Omron Sysmac Studio project Shifting (Sysmac Studio 1.65.0.64007, StandardProject)

# Controller new_Controller_0: NX1P2-1040DT1 version 1.69
Task PrimaryTask (priority 4, period or condition 2000): Program0

VAR_GLOBAL
    IN_Start_But : BOOL;
    IN_Stop_But : BOOL;
    IN_Small_Sens : BOOL;
    IN_Medium_Sens : BOOL;
    IN_High_Sens : BOOL;
    OUT_Konveyor_Start : BOOL;
    OUT_Vana1 : BOOL;
    OUT_Vana2 : BOOL;
    OUT_Vana3 : BOOL;
    OUT_Vana4 : BOOL;
    OUT_Vana5 : BOOL;
    OUT_Vana6 : BOOL;
    OUT_Vana7 : BOOL;
    OUT_Vana8 : BOOL;
    Ary_Bottle : ARRAY[0..8] OF INT;
END_VAR

PROGRAM Program0
VAR
    Start : BOOL;
    Kutu : BOOL;
    Ton_Small : TON;
    medi : BOOL;
    Small_Bottle : BOOL;
    High_Bottle : BOOL;
    Medium_Bottle : BOOL;
    Big_Bottle : BOOL;
    Sayac : INT;
    OUT_Konveyor_Calis : BOOL;
    Konveyor_Calis : BOOL;
    TON_Konv : TON;
    Shiftle : BOOL;
    Small_Bottlei : BOOL;
    TON_Small_Dly : TON;
    TON_Medium_Dly : TON;
    TON_Big_Dly : TON;
    TON_Vana : TON;
    OUT_Vana : BOOL;
    Set_Small : BOOL;
    Set_Medium : BOOL;
    Set_Big : BOOL;
END_VAR
VAR_EXTERNAL
    IN_Start_But : BOOL;
    IN_Stop_But : BOOL;
    IN_Small_Sens : BOOL;
    IN_Medium_Sens : BOOL;
    IN_High_Sens : BOOL;
    OUT_Konveyor_Start : BOOL;
    Ary_Bottle : ARRAY[0..8] OF INT;
    OUT_Vana1 : BOOL;
    OUT_Vana2 : BOOL;
    OUT_Vana3 : BOOL;
    OUT_Vana4 : BOOL;
    OUT_Vana5 : BOOL;
    OUT_Vana6 : BOOL;
    OUT_Vana7 : BOOL;
    OUT_Vana8 : BOOL;
END_VAR
VAR
    _e1 : R_TRIG;
    _e2 : R_TRIG;
    _e3 : R_TRIG;
    _e4 : R_TRIG;
    _e5 : R_TRIG;
    _e6 : R_TRIG;
    _e7 : F_TRIG;
    _e8 : F_TRIG;
    _e9 : F_TRIG;
    _e10 : R_TRIG;
    _e11 : R_TRIG;
    _e12 : R_TRIG;
    _e13 : R_TRIG;
    _e14 : R_TRIG;
    _e15 : R_TRIG;
    _e16 : R_TRIG;
END_VAR

(* Section Section0: ladder, written here as Structured Text *)

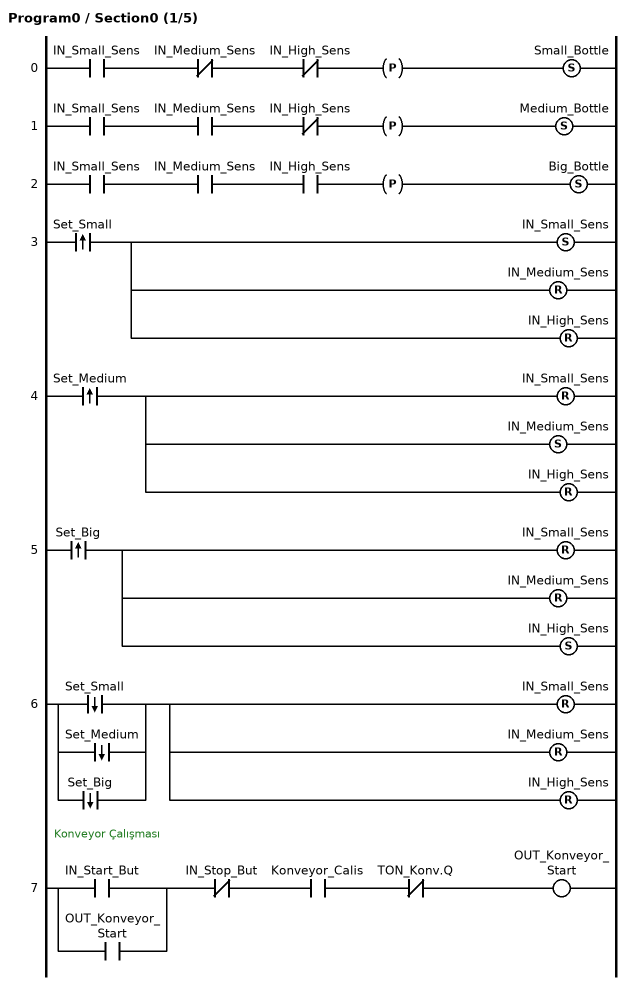
(* Rung 0 *)
_e1(CLK := IN_Small_Sens AND NOT IN_Medium_Sens AND NOT IN_High_Sens);
IF _e1.Q THEN Small_Bottle := TRUE; END_IF;
(* Rung 1 *)
_e2(CLK := IN_Small_Sens AND IN_Medium_Sens AND NOT IN_High_Sens);
IF _e2.Q THEN Medium_Bottle := TRUE; END_IF;
(* Rung 2 *)
_e3(CLK := IN_Small_Sens AND IN_Medium_Sens AND IN_High_Sens);
IF _e3.Q THEN Big_Bottle := TRUE; END_IF;
(* Rung 3 *)
_e4(CLK := Set_Small);
IF _e4.Q THEN
    IN_Small_Sens := TRUE;
    IN_Medium_Sens := FALSE;
    IN_High_Sens := FALSE;
END_IF;
(* Rung 4 *)
_e5(CLK := Set_Medium);
IF _e5.Q THEN
    IN_Small_Sens := FALSE;
    IN_Medium_Sens := TRUE;
    IN_High_Sens := FALSE;
END_IF;
(* Rung 5 *)
_e6(CLK := Set_Big);
IF _e6.Q THEN
    IN_Small_Sens := FALSE;
    IN_Medium_Sens := FALSE;
    IN_High_Sens := TRUE;
END_IF;
(* Rung 6 *)
_e7(CLK := Set_Small);
_e8(CLK := Set_Medium);
_e9(CLK := Set_Big);
IF _e7.Q OR _e8.Q OR _e9.Q THEN
    IN_Small_Sens := FALSE;
    IN_Medium_Sens := FALSE;
    IN_High_Sens := FALSE;
END_IF;
(* Rung 7: Konveyor Çalışması *)
OUT_Konveyor_Start := (IN_Start_But OR OUT_Konveyor_Start) AND NOT IN_Stop_But AND Konveyor_Calis AND NOT TON_Konv.Q;

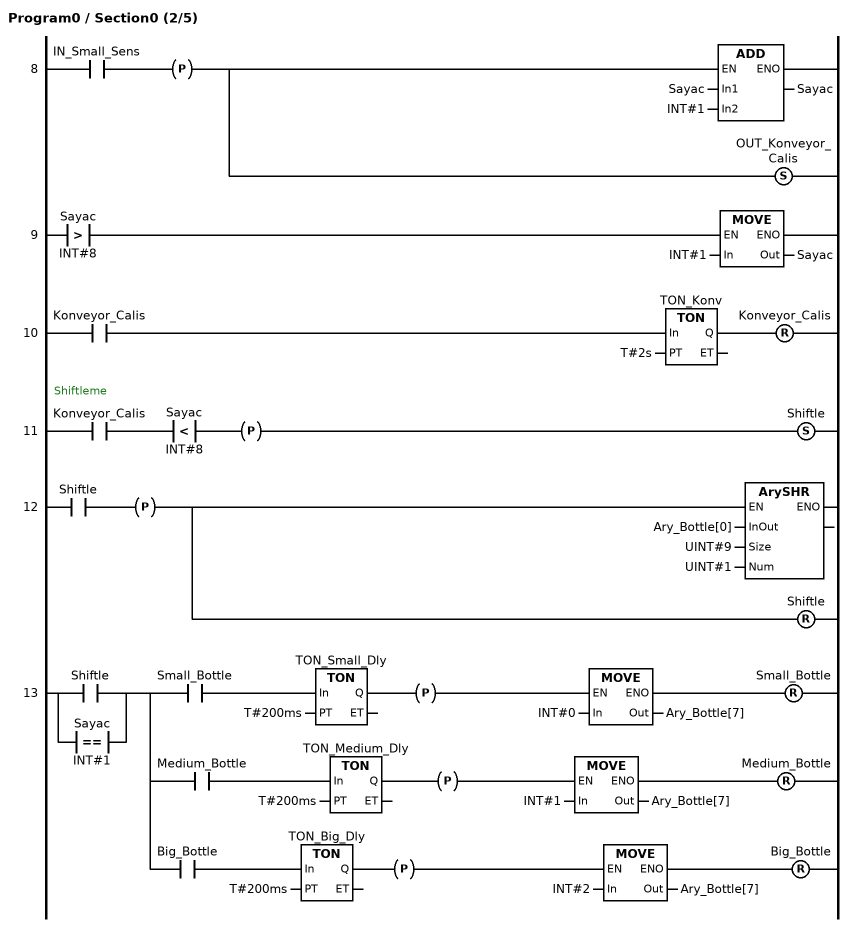
(* Rung 8 *)
_e10(CLK := IN_Small_Sens);
IF _e10.Q THEN
    Sayac := Sayac + INT#1;
    OUT_Konveyor_Calis := TRUE;
END_IF;
(* Rung 9 *)
IF Sayac > INT#8 THEN Sayac := INT#1; END_IF;
(* Rung 10 *)
TON_Konv(In := Konveyor_Calis, PT := T#2s);
IF TON_Konv.Q THEN Konveyor_Calis := FALSE; END_IF;
(* Rung 11: Shiftleme *)
_e11(CLK := Konveyor_Calis AND (Sayac < INT#8));
IF _e11.Q THEN Shiftle := TRUE; END_IF;
(* Rung 12 *)
_e12(CLK := Shiftle);
IF _e12.Q THEN
    ArySHR(InOut := Ary_Bottle[0], Size := UINT#9, Num := UINT#1);
    Shiftle := FALSE;
END_IF;
(* Rung 13 *)
TON_Small_Dly(In := (Shiftle OR (Sayac = INT#1)) AND Small_Bottle, PT := T#200ms);
_e13(CLK := TON_Small_Dly.Q);
IF _e13.Q THEN
    Ary_Bottle[7] := INT#0;
    Small_Bottle := FALSE;
END_IF;
TON_Medium_Dly(In := (Shiftle OR (Sayac = INT#1)) AND Medium_Bottle, PT := T#200ms);
_e14(CLK := TON_Medium_Dly.Q);
IF _e14.Q THEN
    Ary_Bottle[7] := INT#1;
    Medium_Bottle := FALSE;
END_IF;
TON_Big_Dly(In := (Shiftle OR (Sayac = INT#1)) AND Big_Bottle, PT := T#200ms);
_e15(CLK := TON_Big_Dly.Q);
IF _e15.Q THEN
    Ary_Bottle[7] := INT#2;
    Big_Bottle := FALSE;
END_IF;

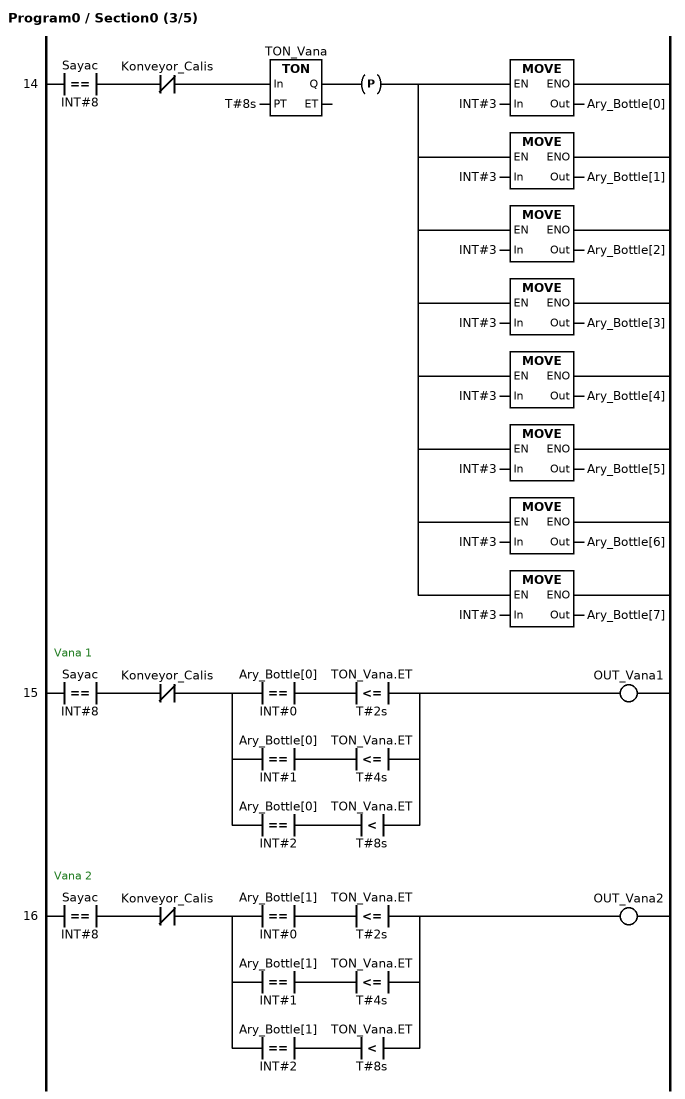
(* Rung 14 *)
TON_Vana(In := (Sayac = INT#8) AND NOT Konveyor_Calis, PT := T#8s);
_e16(CLK := TON_Vana.Q);
IF _e16.Q THEN
    Ary_Bottle[0] := INT#3;
    Ary_Bottle[1] := INT#3;
    Ary_Bottle[2] := INT#3;
    Ary_Bottle[3] := INT#3;
    Ary_Bottle[4] := INT#3;
    Ary_Bottle[5] := INT#3;
    Ary_Bottle[6] := INT#3;
    Ary_Bottle[7] := INT#3;
END_IF;
(* Rung 15: Vana 1 *)
OUT_Vana1 := (Sayac = INT#8) AND NOT Konveyor_Calis AND (((Ary_Bottle[0] = INT#0) AND (TON_Vana.ET <= T#2s)) OR ((Ary_Bottle[0] = INT#1) AND (TON_Vana.ET <= T#4s)) OR ((Ary_Bottle[0] = INT#2) AND (TON_Vana.ET < T#8s)));
(* Rung 16: Vana 2 *)
OUT_Vana2 := (Sayac = INT#8) AND NOT Konveyor_Calis AND (((Ary_Bottle[1] = INT#0) AND (TON_Vana.ET <= T#2s)) OR ((Ary_Bottle[1] = INT#1) AND (TON_Vana.ET <= T#4s)) OR ((Ary_Bottle[1] = INT#2) AND (TON_Vana.ET < T#8s)));

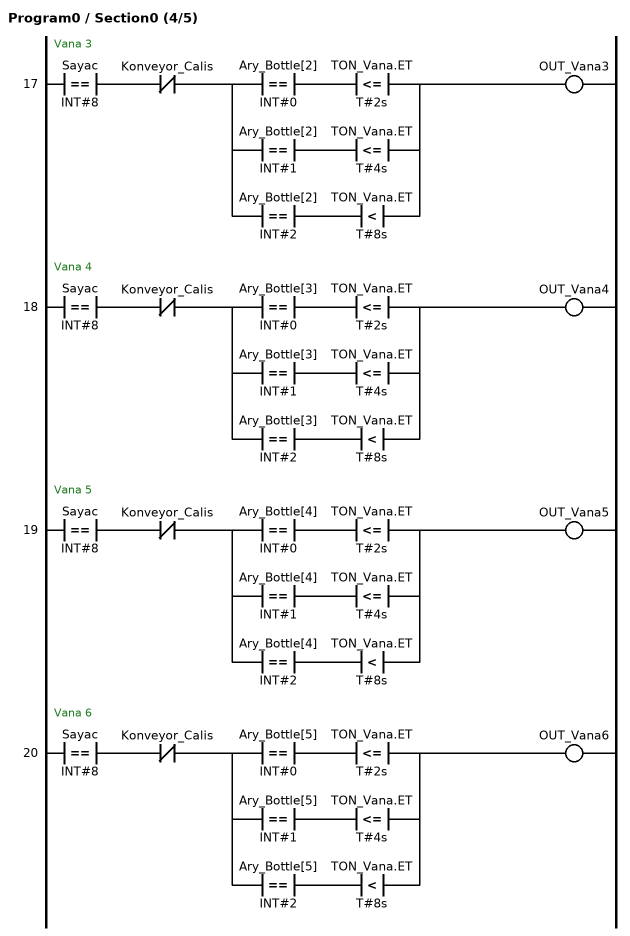
(* Rung 17: Vana 3 *)
OUT_Vana3 := (Sayac = INT#8) AND NOT Konveyor_Calis AND (((Ary_Bottle[2] = INT#0) AND (TON_Vana.ET <= T#2s)) OR ((Ary_Bottle[2] = INT#1) AND (TON_Vana.ET <= T#4s)) OR ((Ary_Bottle[2] = INT#2) AND (TON_Vana.ET < T#8s)));
(* Rung 18: Vana 4 *)
OUT_Vana4 := (Sayac = INT#8) AND NOT Konveyor_Calis AND (((Ary_Bottle[3] = INT#0) AND (TON_Vana.ET <= T#2s)) OR ((Ary_Bottle[3] = INT#1) AND (TON_Vana.ET <= T#4s)) OR ((Ary_Bottle[3] = INT#2) AND (TON_Vana.ET < T#8s)));
(* Rung 19: Vana 5 *)
OUT_Vana5 := (Sayac = INT#8) AND NOT Konveyor_Calis AND (((Ary_Bottle[4] = INT#0) AND (TON_Vana.ET <= T#2s)) OR ((Ary_Bottle[4] = INT#1) AND (TON_Vana.ET <= T#4s)) OR ((Ary_Bottle[4] = INT#2) AND (TON_Vana.ET < T#8s)));
(* Rung 20: Vana 6 *)
OUT_Vana6 := (Sayac = INT#8) AND NOT Konveyor_Calis AND (((Ary_Bottle[5] = INT#0) AND (TON_Vana.ET <= T#2s)) OR ((Ary_Bottle[5] = INT#1) AND (TON_Vana.ET <= T#4s)) OR ((Ary_Bottle[5] = INT#2) AND (TON_Vana.ET < T#8s)));

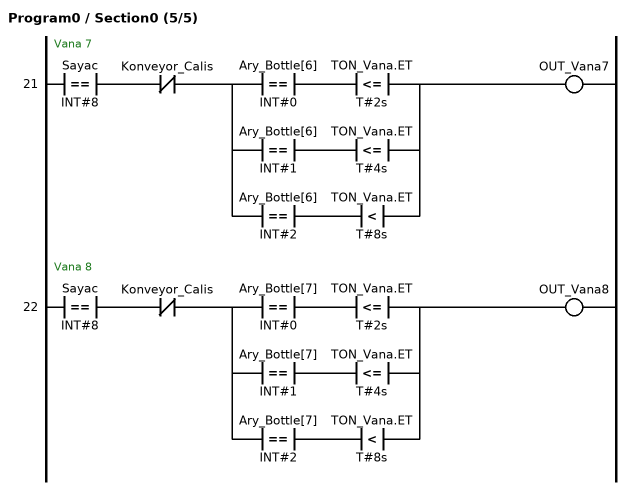
(* Rung 21: Vana 7 *)
OUT_Vana7 := (Sayac = INT#8) AND NOT Konveyor_Calis AND (((Ary_Bottle[6] = INT#0) AND (TON_Vana.ET <= T#2s)) OR ((Ary_Bottle[6] = INT#1) AND (TON_Vana.ET <= T#4s)) OR ((Ary_Bottle[6] = INT#2) AND (TON_Vana.ET < T#8s)));
(* Rung 22: Vana 8 *)
OUT_Vana8 := (Sayac = INT#8) AND NOT Konveyor_Calis AND (((Ary_Bottle[7] = INT#0) AND (TON_Vana.ET <= T#2s)) OR ((Ary_Bottle[7] = INT#1) AND (TON_Vana.ET <= T#4s)) OR ((Ary_Bottle[7] = INT#2) AND (TON_Vana.ET < T#8s)));
END_PROGRAM